{attribute addProperty BoxType "EK1100-0000-0018"}
{attribute addProperty Id "Beckhoff_EL5xxxEK1122Beckhoff_EL5xxxEK1122_F18478E1162A_0001_EL5001_0000_0000EL5001_9629689812215.25A_0002_EL5001_0000_0001EL5001_9629689812215.25A_0003_EL5001_0000_1016EL5001_C393BC8012215.25A_0004_EL5001_0000_1017EL5001_2283773F13016.25A_0005_EL5001_0000_1018EL5001_2283773F13016.25A_0006_EL5001_0000_1019EL5001_2283773F13016.25A_0007_EL5001_0000_1020EL5001_2283773F13016.25A_0008_EL5001_0000_1021EL5001_0BD730D013016.25A_0009_EL5001_0010_0000EL5001_9629689812215.25A_0010_EL5001_0011_0016EL5001_F5F6E71822628.25A_0011_EL5001_0011_0017EL5001_F5F6E71822628.25A_0012_EL5001_0011_0018EL5001_F5F6E71822628.25A_0013_EL5001_0011_0019EL5001_09B94A5B19424.25A_0014_EL5001_0011_0020EL5001_09B94A5B19424.25A_0015_EL5001_0090_0016EL5001_99FC62FA13016.25A_0016_EL5002_0000_0016EL5002_8228306817822.25A_0017_EL5002_0000_0017EL5002_8228306817822.25A_0018_EL5002_0000_0018EL5002_8228306817822.25A_0019_EL5002_0000_0019EL5002_8228306817822.25A_0020_EL5002_0000_0020EL5002_960CC6F117822.25A_0021_EL5021_0000_0016EL5021_32D1A2A321026.25A_0022_EL5021_0000_0017EL5021_32D1A2A321026.25A_0023_EL5021_0000_0018EL5021_32D1A2A321026.25A_0024_EL5021_0000_0019EL5021_1B8188B721026.25A_0025_EL5021_0000_0020EL5021_1B8188B721026.25A_0026_EL5021_0000_0021EL5021_1B8188B721026.25A_0027_EL5021_0000_0022EL5021_1B8188B721026.25A_0028_EL5021_0090_0018EL5021_1B8188B721026.25A_0029_EL5021_0090_0019EL5021_1B8188B721026.25A_0030_EL5032_0000_0021EL5032_3D8BD04C24230.25A_0031_EL5032_0000_0023EL5032_3D8BD04C24230.25A_0032_EL5032_0000_0024EL5032_3D8BD04C24230.25A_0033_EL5032_0000_0025EL5032_3D8BD04C24230.25A_0034_EL5032_0000_0026EL5032_3D8BD04C24230.25A_0035_EL5032_0000_0027EL5032_3D8BD04C24230.25A_0036_EL5032_0090_0016EL5032_3D8BD04C24230.25A_0037_EL5042_0000_0016EL5042_3D8BD04C24230.25A_0038_EL5072_0000_0016EL5072_762C412B35444.25A_0039_EL5101_0000_0000EL5101_8E82486614618.25A_0040_EL5101_0000_0001EL5101_38C6EF5E14618.25A_0041_EL5101_0000_1017EL5101_38C6EF5E14618.25A_0042_EL5101_0000_1018EL5101_38C6EF5E14618.25A_0043_EL5101_0000_1019EL5101_2133D81029036.25A_0044_EL5101_0000_1020EL5101_5EFFFA4516220.25A_0045_EL5101_0000_1021EL5101_5EFFFA4516220.25A_0046_EL5101_0000_1022EL5101_5EFFFA4516220.25A_0047_EL5101_0000_1023EL5101_6012872616220.25A_0048_EL5101_0000_1024EL5101_6012872616220.25A_0049_EL5101_0010_0016EL5101_1151690E16220.25A_0050_EL5101_0010_0017EL5101_1151690E16220.25A_0051_EL5101_0010_0018EL5101_1151690E16220.25A_0052_EL5101_0010_0019EL5101_354B248916220.25A_0053_EL5101_0011_0016EL5101_28E4060930638.25A_0054_EL5101_0090_0016EL5101_6012872616220.25A_0055_EL5101_0090_0017EL5101_6012872616220.25A_0056_EL5101_1006_1019EL5101_2133D81029036.25A_0057_EL5101_1006_1020EL5101_5EFFFA4516220.25A_0058_EL5101_1006_1021EL5101_5EFFFA4516220.25A_0059_EL5101_1006_1022EL5101_5EFFFA4516220.25A_0060_EL5101_1006_1023EL5101_5EFFFA4516220.25A_0061_EL5151_0000_0016EL5151_7DE9C09925832.25A_0062_EL5102_0000_0016EL5102_C51BD5F643454.25A_0063_EL5112_0000_0016EL5112_3D3BC26F25832.25A_0064_EL5122_0000_0016EL5122_D4BE45F537046.25A_0065_EL5151_0000_0017EL5151_023DC4F232240.25A_0066_EL5151_0000_0018EL5151_023DC4F232240.25A_0067_EL5151_0000_0019EL5151_023DC4F232240.25A_0068_EL5151_0000_0020EL5151_B6C9029519424.25A_0069_EL5151_0000_0021EL5151_1872592219424.25A_0070_EL5151_0000_0022EL5151_1872592219424.25A_0071_EL5151_0000_0023EL5151_1872592219424.25A_0072_EL5151_0000_0024EL5151_1872592219424.25A_0073_EL5151_0000_0025EL5151_0AC1A36D19424.25A_0074_EL5151_0000_0026EL5151_0AC1A36D19424.25A_0075_EL5151_0021_0018EL5151_0683EF8C33842.25A_0076_EL5151_0080_0016EL5151_09E56EF027434.25A_0077_EL5151_0080_0017EL5151_B6C9029519424.25A_0078_EL5151_0080_0018EL5151_B6C9029519424.25A_0079_EL5151_0080_0019EL5151_B6C9029519424.25A_0080_EL5151_0080_0020EL5151_B6C9029519424.25A_0081_EL5151_0080_0021EL5151_0AC1A36D19424.25A_0082_EL5151_0090_0016EL5151_8E09C6BA16220.25A_0083_EL5152_0000_0016EL5152_A669F51732240.25A_0084_EL5152_0000_0017EL5152_A669F51732240.25A_0085_EL5152_0000_0018EL5152_9ECEB73927434.25A_0086_EL5152_0000_0019EL5152_9ECEB73927434.25"}
{attribute addProperty CRC "3356208894"}
{attribute addProperty SizeInBites "17900"}
{attribute addProperty SizeInBytes "2237.5"}
TYPE Beckhoff_EL5xxx_C80BAEFE EXTENDS EK1100_179A0949 :
STRUCT
	{attribute addProperty Name "Beckhoff_EL5xxxEK1122"}
	Beckhoff_EL5xxxEK1122 : Beckhoff_EL5xxxEK1122_F18478E1;
	{attribute addProperty Name "A_0001_EL5001_0000_0000"}
	A_0001_EL5001_0000_0000 : EL5001_96296898;
	{attribute addProperty Name "A_0002_EL5001_0000_0001"}
	A_0002_EL5001_0000_0001 : EL5001_96296898;
	{attribute addProperty Name "A_0003_EL5001_0000_1016"}
	A_0003_EL5001_0000_1016 : EL5001_C393BC80;
	{attribute addProperty Name "A_0004_EL5001_0000_1017"}
	A_0004_EL5001_0000_1017 : EL5001_2283773F;
	{attribute addProperty Name "A_0005_EL5001_0000_1018"}
	A_0005_EL5001_0000_1018 : EL5001_2283773F;
	{attribute addProperty Name "A_0006_EL5001_0000_1019"}
	A_0006_EL5001_0000_1019 : EL5001_2283773F;
	{attribute addProperty Name "A_0007_EL5001_0000_1020"}
	A_0007_EL5001_0000_1020 : EL5001_2283773F;
	{attribute addProperty Name "A_0008_EL5001_0000_1021"}
	A_0008_EL5001_0000_1021 : EL5001_0BD730D0;
	{attribute addProperty Name "A_0009_EL5001_0010_0000"}
	A_0009_EL5001_0010_0000 : EL5001_96296898;
	{attribute addProperty Name "A_0010_EL5001_0011_0016"}
	A_0010_EL5001_0011_0016 : EL5001_F5F6E718;
	{attribute addProperty Name "A_0011_EL5001_0011_0017"}
	A_0011_EL5001_0011_0017 : EL5001_F5F6E718;
	{attribute addProperty Name "A_0012_EL5001_0011_0018"}
	A_0012_EL5001_0011_0018 : EL5001_F5F6E718;
	{attribute addProperty Name "A_0013_EL5001_0011_0019"}
	A_0013_EL5001_0011_0019 : EL5001_09B94A5B;
	{attribute addProperty Name "A_0014_EL5001_0011_0020"}
	A_0014_EL5001_0011_0020 : EL5001_09B94A5B;
	{attribute addProperty Name "A_0015_EL5001_0090_0016"}
	A_0015_EL5001_0090_0016 : EL5001_99FC62FA;
	{attribute addProperty Name "A_0016_EL5002_0000_0016"}
	A_0016_EL5002_0000_0016 : EL5002_82283068;
	{attribute addProperty Name "A_0017_EL5002_0000_0017"}
	A_0017_EL5002_0000_0017 : EL5002_82283068;
	{attribute addProperty Name "A_0018_EL5002_0000_0018"}
	A_0018_EL5002_0000_0018 : EL5002_82283068;
	{attribute addProperty Name "A_0019_EL5002_0000_0019"}
	A_0019_EL5002_0000_0019 : EL5002_82283068;
	{attribute addProperty Name "A_0020_EL5002_0000_0020"}
	A_0020_EL5002_0000_0020 : EL5002_960CC6F1;
	{attribute addProperty Name "A_0021_EL5021_0000_0016"}
	A_0021_EL5021_0000_0016 : EL5021_32D1A2A3;
	{attribute addProperty Name "A_0022_EL5021_0000_0017"}
	A_0022_EL5021_0000_0017 : EL5021_32D1A2A3;
	{attribute addProperty Name "A_0023_EL5021_0000_0018"}
	A_0023_EL5021_0000_0018 : EL5021_32D1A2A3;
	{attribute addProperty Name "A_0024_EL5021_0000_0019"}
	A_0024_EL5021_0000_0019 : EL5021_1B8188B7;
	{attribute addProperty Name "A_0025_EL5021_0000_0020"}
	A_0025_EL5021_0000_0020 : EL5021_1B8188B7;
	{attribute addProperty Name "A_0026_EL5021_0000_0021"}
	A_0026_EL5021_0000_0021 : EL5021_1B8188B7;
	{attribute addProperty Name "A_0027_EL5021_0000_0022"}
	A_0027_EL5021_0000_0022 : EL5021_1B8188B7;
	{attribute addProperty Name "A_0028_EL5021_0090_0018"}
	A_0028_EL5021_0090_0018 : EL5021_1B8188B7;
	{attribute addProperty Name "A_0029_EL5021_0090_0019"}
	A_0029_EL5021_0090_0019 : EL5021_1B8188B7;
	{attribute addProperty Name "A_0030_EL5032_0000_0021"}
	A_0030_EL5032_0000_0021 : EL5032_3D8BD04C;
	{attribute addProperty Name "A_0031_EL5032_0000_0023"}
	A_0031_EL5032_0000_0023 : EL5032_3D8BD04C;
	{attribute addProperty Name "A_0032_EL5032_0000_0024"}
	A_0032_EL5032_0000_0024 : EL5032_3D8BD04C;
	{attribute addProperty Name "A_0033_EL5032_0000_0025"}
	A_0033_EL5032_0000_0025 : EL5032_3D8BD04C;
	{attribute addProperty Name "A_0034_EL5032_0000_0026"}
	A_0034_EL5032_0000_0026 : EL5032_3D8BD04C;
	{attribute addProperty Name "A_0035_EL5032_0000_0027"}
	A_0035_EL5032_0000_0027 : EL5032_3D8BD04C;
	{attribute addProperty Name "A_0036_EL5032_0090_0016"}
	A_0036_EL5032_0090_0016 : EL5032_3D8BD04C;
	{attribute addProperty Name "A_0037_EL5042_0000_0016"}
	A_0037_EL5042_0000_0016 : EL5042_3D8BD04C;
	{attribute addProperty Name "A_0038_EL5072_0000_0016"}
	A_0038_EL5072_0000_0016 : EL5072_762C412B;
	{attribute addProperty Name "A_0039_EL5101_0000_0000"}
	A_0039_EL5101_0000_0000 : EL5101_8E824866;
	{attribute addProperty Name "A_0040_EL5101_0000_0001"}
	A_0040_EL5101_0000_0001 : EL5101_38C6EF5E;
	{attribute addProperty Name "A_0041_EL5101_0000_1017"}
	A_0041_EL5101_0000_1017 : EL5101_38C6EF5E;
	{attribute addProperty Name "A_0042_EL5101_0000_1018"}
	A_0042_EL5101_0000_1018 : EL5101_38C6EF5E;
	{attribute addProperty Name "A_0043_EL5101_0000_1019"}
	A_0043_EL5101_0000_1019 : EL5101_2133D810;
	{attribute addProperty Name "A_0044_EL5101_0000_1020"}
	A_0044_EL5101_0000_1020 : EL5101_5EFFFA45;
	{attribute addProperty Name "A_0045_EL5101_0000_1021"}
	A_0045_EL5101_0000_1021 : EL5101_5EFFFA45;
	{attribute addProperty Name "A_0046_EL5101_0000_1022"}
	A_0046_EL5101_0000_1022 : EL5101_5EFFFA45;
	{attribute addProperty Name "A_0047_EL5101_0000_1023"}
	A_0047_EL5101_0000_1023 : EL5101_60128726;
	{attribute addProperty Name "A_0048_EL5101_0000_1024"}
	A_0048_EL5101_0000_1024 : EL5101_60128726;
	{attribute addProperty Name "A_0049_EL5101_0010_0016"}
	A_0049_EL5101_0010_0016 : EL5101_1151690E;
	{attribute addProperty Name "A_0050_EL5101_0010_0017"}
	A_0050_EL5101_0010_0017 : EL5101_1151690E;
	{attribute addProperty Name "A_0051_EL5101_0010_0018"}
	A_0051_EL5101_0010_0018 : EL5101_1151690E;
	{attribute addProperty Name "A_0052_EL5101_0010_0019"}
	A_0052_EL5101_0010_0019 : EL5101_354B2489;
	{attribute addProperty Name "A_0053_EL5101_0011_0016"}
	A_0053_EL5101_0011_0016 : EL5101_28E40609;
	{attribute addProperty Name "A_0054_EL5101_0090_0016"}
	A_0054_EL5101_0090_0016 : EL5101_60128726;
	{attribute addProperty Name "A_0055_EL5101_0090_0017"}
	A_0055_EL5101_0090_0017 : EL5101_60128726;
	{attribute addProperty Name "A_0056_EL5101_1006_1019"}
	A_0056_EL5101_1006_1019 : EL5101_2133D810;
	{attribute addProperty Name "A_0057_EL5101_1006_1020"}
	A_0057_EL5101_1006_1020 : EL5101_5EFFFA45;
	{attribute addProperty Name "A_0058_EL5101_1006_1021"}
	A_0058_EL5101_1006_1021 : EL5101_5EFFFA45;
	{attribute addProperty Name "A_0059_EL5101_1006_1022"}
	A_0059_EL5101_1006_1022 : EL5101_5EFFFA45;
	{attribute addProperty Name "A_0060_EL5101_1006_1023"}
	A_0060_EL5101_1006_1023 : EL5101_5EFFFA45;
	{attribute addProperty Name "A_0061_EL5151_0000_0016"}
	A_0061_EL5151_0000_0016 : EL5151_7DE9C099;
	{attribute addProperty Name "A_0062_EL5102_0000_0016"}
	A_0062_EL5102_0000_0016 : EL5102_C51BD5F6;
	{attribute addProperty Name "A_0063_EL5112_0000_0016"}
	A_0063_EL5112_0000_0016 : EL5112_3D3BC26F;
	{attribute addProperty Name "A_0064_EL5122_0000_0016"}
	A_0064_EL5122_0000_0016 : EL5122_D4BE45F5;
	{attribute addProperty Name "A_0065_EL5151_0000_0017"}
	A_0065_EL5151_0000_0017 : EL5151_023DC4F2;
	{attribute addProperty Name "A_0066_EL5151_0000_0018"}
	A_0066_EL5151_0000_0018 : EL5151_023DC4F2;
	{attribute addProperty Name "A_0067_EL5151_0000_0019"}
	A_0067_EL5151_0000_0019 : EL5151_023DC4F2;
	{attribute addProperty Name "A_0068_EL5151_0000_0020"}
	A_0068_EL5151_0000_0020 : EL5151_B6C90295;
	{attribute addProperty Name "A_0069_EL5151_0000_0021"}
	A_0069_EL5151_0000_0021 : EL5151_18725922;
	{attribute addProperty Name "A_0070_EL5151_0000_0022"}
	A_0070_EL5151_0000_0022 : EL5151_18725922;
	{attribute addProperty Name "A_0071_EL5151_0000_0023"}
	A_0071_EL5151_0000_0023 : EL5151_18725922;
	{attribute addProperty Name "A_0072_EL5151_0000_0024"}
	A_0072_EL5151_0000_0024 : EL5151_18725922;
	{attribute addProperty Name "A_0073_EL5151_0000_0025"}
	A_0073_EL5151_0000_0025 : EL5151_0AC1A36D;
	{attribute addProperty Name "A_0074_EL5151_0000_0026"}
	A_0074_EL5151_0000_0026 : EL5151_0AC1A36D;
	{attribute addProperty Name "A_0075_EL5151_0021_0018"}
	A_0075_EL5151_0021_0018 : EL5151_0683EF8C;
	{attribute addProperty Name "A_0076_EL5151_0080_0016"}
	A_0076_EL5151_0080_0016 : EL5151_09E56EF0;
	{attribute addProperty Name "A_0077_EL5151_0080_0017"}
	A_0077_EL5151_0080_0017 : EL5151_B6C90295;
	{attribute addProperty Name "A_0078_EL5151_0080_0018"}
	A_0078_EL5151_0080_0018 : EL5151_B6C90295;
	{attribute addProperty Name "A_0079_EL5151_0080_0019"}
	A_0079_EL5151_0080_0019 : EL5151_B6C90295;
	{attribute addProperty Name "A_0080_EL5151_0080_0020"}
	A_0080_EL5151_0080_0020 : EL5151_B6C90295;
	{attribute addProperty Name "A_0081_EL5151_0080_0021"}
	A_0081_EL5151_0080_0021 : EL5151_0AC1A36D;
	{attribute addProperty Name "A_0082_EL5151_0090_0016"}
	A_0082_EL5151_0090_0016 : EL5151_8E09C6BA;
	{attribute addProperty Name "A_0083_EL5152_0000_0016"}
	A_0083_EL5152_0000_0016 : EL5152_A669F517;
	{attribute addProperty Name "A_0084_EL5152_0000_0017"}
	A_0084_EL5152_0000_0017 : EL5152_A669F517;
	{attribute addProperty Name "A_0085_EL5152_0000_0018"}
	A_0085_EL5152_0000_0018 : EL5152_9ECEB739;
	{attribute addProperty Name "A_0086_EL5152_0000_0019"}
	A_0086_EL5152_0000_0019 : EL5152_9ECEB739;
END_STRUCT
END_TYPE

(* stored: Version 1.2.0.0, ProductVersion 3.1.4024.9
   DUT Beckhoff_EL5xxx_C80BAEFE: Id {88a66218-8c3d-4806-aefa-cbc3f7fd7ede} *)
